// TIA Portal V17 export
// export: Created 2023-12-22T15:28:37.6309376Z, ExportSetting WithDefaults, DisplayName Totally Integrated Automation Portal, DisplayVersion V17, DisplayName TIA Portal Openness, DisplayVersion V17, DisplayName TIA Portal Version Control Interface, DisplayVersion V17, DisplayName STEP 7 Professional, DisplayVersion V17, DisplayName STEP 7 Safety, DisplayVersion V17, DisplayName WinCC Advanced, DisplayVersion V17
DATA_BLOCK "ModBus_RTU_DB"   // DB30
VERSION : 0.1
// stored: AutoNumber false, DBAccessibleFromOPCUA true, InstanceOfName ModBus_RTU, InstanceOfType FB
"ModBus_RTU"
   // VAR RETAIN
   //    DATA : Array[0..100] of Word;
   //    "Step" : Int;
   //    Device : Int;
   //    Limit { S7_SetPoint := 'True'} : Int;
   //    COM_Config : Struct
   //       Baud_Rate { S7_SetPoint := 'True'} : UDInt;
   //       Port { S7_SetPoint := 'True'} : PORT;
   //    END_STRUCT;
   //    COM_Control : Struct
   //       Enable { S7_SetPoint := 'True'} : Bool;
   //       Start : Bool;
   //       Reset : Bool;
   //       Load_Done : Bool;
   //       Load_Status : Word;
   //       REQ_Done : Bool;
   //       REQ_Busy : Bool;
   //       REQ_Error : Bool;
   //       REQ_Status : Word;
   //       Error_Code : Word;
   //       Status : Int;
   //    END_STRUCT;
   //    COM_REQ : Struct
   //       ADDR : UInt;
   //       MODE : USInt;
   //       Register : UDInt;
   //       Length : UInt;
   //    END_STRUCT;
   //    DEV_Config : Array[1..10] of Struct
   //       Use { S7_SetPoint := 'True'} : Bool;
   //       MODE { S7_SetPoint := 'True'} : Bool;
   //       ADDR { S7_SetPoint := 'True'} : UInt;
   //       Register { S7_SetPoint := 'True'} : UDInt;
   //       Length { S7_SetPoint := 'True'} : UInt;
   //       Source_DB { S7_SetPoint := 'True'} : UInt;
   //       Source_OFFSET { S7_SetPoint := 'True'} : UInt;
   //       Target_DB { S7_SetPoint := 'True'} : UInt;
   //       Target_OFFSET { S7_SetPoint := 'True'} : UInt;
   //       Status : UInt;
   //    END_STRUCT;
   //    MB_COMM_LOAD : MB_COMM_LOAD;
   //    MB_MASTER : MB_MASTER;
   //    T_Busy : "Time_M";
   // END_VAR
BEGIN
END_DATA_BLOCK
